// LS Electric XG5000 project: 0211_LS_MODBUS
// PLC NewPLC

PROGRAM Main (task: 스캔 프로그램)

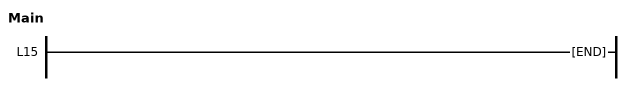
; L15
END